Fanuc KAREL source: kt00333.KL

-- PROVISIONAL review KL for V1013-1; original PC SHA256 849e348906ef1172fd9e367efaf31683dc4c471815d68edcd4d8839f6fb6236f
-- Incomplete behavior may be omitted. Consult companion uncertainty JSON. Do not deploy.
PROGRAM KT00333
%NOLOCKGROUP
VAR
  R1 : REAL
  I2 : INTEGER
  OUT : BOOLEAN
BEGIN
  -- UNRESOLVED_PC offsets 5-16; opcodes 2E,23
  -- UNRESOLVED_PC offsets 21-32; opcodes 2E,23
  -- UNRESOLVED_PC offsets 37-57; opcodes 21,21,64,6F,23
  -- UNRESOLVED_PC offsets 62-66; opcodes 7F
END KT00333
